# B&R Automation Studio project B-R-lab1
Automation Studio 4.5.2.102

## Configuration Config1

CPU 4PP065.0571-P74, AutomationRuntime D4.52, Build 4.1.2, Vc V4.52.0

### Hardware
```
4PP065_0571_P74 : 4PP065.0571-P74 v1.2.0.0
  Connector IF4:
    DNAConfiguration = manual
  Connector IF5:
    ActivateDevice = 1
    Mode = Manual
    InternetAddress = 10.0.1.10
    SubnetMask = 255.255.255.0
  ConfigurationID = labBR
  Simulation = 1
  Cyclic3Duration = 40000
  Cyclic3Tolerance = 40000
```

## Logical view

Binary libraries used (declarations not repeated): operator, runtime, astime, AsIecCon

### Library Logical/Libraries/Coollb (ANSIC)

#### Constants.var - Exported constants
```iecst
VAR CONSTANT
	d_t : REAL := 0.01;
END_VAR
```

#### Coollb.fun - Exported functions and function blocks
```iecst
{REDUND_ERROR} FUNCTION_BLOCK FB_Motor (*TODO: Add your comment here*) (*$GROUP=User,$CAT=User,$GROUPICON=User.png,$CATICON=User.png*)
	VAR_INPUT
		u : {REDUND_UNREPLICABLE} REAL;
	END_VAR
	VAR_OUTPUT
		w : {REDUND_UNREPLICABLE} REAL;
		phi : {REDUND_UNREPLICABLE} REAL;
	END_VAR
	VAR
		integrator : {REDUND_UNREPLICABLE} FB_Integrator;
		Tm : {REDUND_UNREPLICABLE} REAL;
		ke : {REDUND_UNREPLICABLE} REAL;
	END_VAR
	VAR_INPUT
		dt : REAL;
	END_VAR
END_FUNCTION_BLOCK

FUNCTION_BLOCK FB_Integrator
	VAR_INPUT
		in : {REDUND_UNREPLICABLE} REAL;
		dt : REAL;
	END_VAR
	VAR_OUTPUT
		out : {REDUND_UNREPLICABLE} REAL;
	END_VAR
	VAR
		prev_value : REAL;
	END_VAR
END_FUNCTION_BLOCK

FUNCTION_BLOCK FB_Controller
	VAR_INPUT
		e_in : {REDUND_UNREPLICABLE} REAL;
	END_VAR
	VAR_OUTPUT
		u_out : {REDUND_UNREPLICABLE} REAL;
	END_VAR
	VAR
		sum : REAL;
		a : REAL;
		k_p : REAL;
		k_i : REAL;
	END_VAR
	VAR_INPUT
		dt : REAL;
	END_VAR
	VAR
		max_abs_value : REAL;
		iyOld : REAL;
		integrator : FB_Integrator;
		last_sum : REAL;
	END_VAR
END_FUNCTION_BLOCK
```

#### FB_motor.c
```c
#include <bur/plctypes.h>
#ifdef __cplusplus
	extern "C"
	{
#endif
	#include "Coollb.h"
#ifdef __cplusplus
	};
#endif
/* TODO: Add your comment here */
void FB_Motor(struct FB_Motor* inst)
{
	REAL a = (inst->u/inst->ke) - inst->w;
	REAL b = a / inst->Tm;

	inst->integrator.in = b;
	FB_Integrator(&inst->integrator);

	inst->w = inst->integrator.out;

	inst->integrator.in = inst->w;
	FB_Integrator(&inst->integrator);

	inst->phi = inst->integrator.out;

}
```

#### FB_Integrator.c
```c
#include <bur/plctypes.h>
#ifdef __cplusplus
	extern "C"
	{
#endif
	#include "Coollb.h"
#ifdef __cplusplus
	};
#endif
/* TODO: Add your comment here */
void FB_Integrator(struct FB_Integrator* inst)
{
	inst->dt = d_t;
	inst->out = inst->dt * inst->in + inst->prev_value;
	inst->prev_value = inst->out;
}
```

#### FB_Controller.c
```c
#include <bur/plctypes.h>
#ifdef __cplusplus
	extern "C"
	{
#endif
	#include "Coollb.h"
#ifdef __cplusplus
	};
#endif
/* TODO: Add your comment here */
void FB_Controller(struct FB_Controller* inst)
{
	REAL a = inst->e_in * inst->k_p;
	REAL b = inst->e_in * inst->k_i;

	a = a > inst->max_abs_value ? inst->max_abs_value : a;
	a = a < -inst->max_abs_value ? -inst->max_abs_value : a;

	inst->integrator.in = b + inst->last_sum;
	FB_Integrator(&inst->integrator);

	REAL sum = a + inst->integrator.out;

	inst->u_out = sum;//inst->u_out = inst->a

	inst->u_out = inst->u_out > inst->max_abs_value ? inst->max_abs_value : inst->u_out;
	inst->u_out = inst->u_out < -inst->max_abs_value ? -inst->max_abs_value : inst->u_out;

	inst->last_sum = inst->u_out - sum; //inst->iyOld = inst->u_out - sum;

}
```

### Program Logical/Program

#### Variables.var
```iecst
VAR
	enable : BOOL;
	counter : UINT;
	speed : REAL;
	fb_motor2 : FB_Motor;
	fb_motor1 : FB_Motor;
	fb_controller : FB_Controller;
END_VAR
```

#### Main.c
```c
#include <bur/plctypes.h>

#ifdef _DEFAULT_INCLUDES
	#include <AsDefault.h>
#endif

void _INIT ProgramInit(void)
{
	/*
	ke = 0.24
	Tm = 0.1

	k_p = 0.78
	k_i = 7.2

	наш двигун

	ke = 0.181
	Tm = 0.25

	k_p = 0.6525
	k_i = 2.0

	*/
	fb_motor1.ke = 0.24;
	fb_motor1.Tm = 0.1;
	fb_motor1.u = 0;

	fb_motor2.ke = 0.181;
	fb_motor2.Tm = 0.25;
	fb_motor2.u = 0;

	fb_controller.k_p = 0.78;
	fb_controller.k_i = 7.2;
	fb_controller.max_abs_value = 24.0;//24

	speed = 0;
	counter = 0;
	enable = 0;
}

void _CYCLIC ProgramCyclic(void)
{
	if(enable)
	{
		if(counter == 200)
		{
			speed = 0;
			counter = 0;
		}
		else if (counter == 50)
		{
			speed = 50;
		}

		fb_controller.e_in = speed - fb_motor1.w;
		FB_Controller(&fb_controller);

		fb_motor1.u = fb_controller.u_out;
		FB_Motor(&fb_motor1);

		fb_motor2.u = speed * fb_motor2.ke;
		FB_Motor(&fb_motor2);

		counter++;
	}
	else
	{
		speed = 0;
		counter = 0;
	}
}

void _EXIT ProgramExit(void)
{

}
```

Listed in the project but not available here: Logical/Libraries/Coollb/Types.typ
